Fanuc KAREL source: kt00901.KL

PROGRAM KT00901
%STACKSIZE=65535
%PRIORITY=65535
%NOLOCKGROUP
VAR
P1 : JOINTPOS9
P2 : JOINTPOS9
OUT : BOOLEAN
BEGIN
-- UNRESOLVED_PC line 8 opcodes [27 22 1C 27 9D 76 23] marker_code=0
END KT00901
